// TIA Portal project "Software Units Example - Stack" (V17)

(* hardware
DEVICE "S7-1500/ET200MP station_1"  S7-1500 station
   slot 0: "Rail_0"  Rack  6ES7 590-1***0-0AA0
   slot 1: "PLC_1"  CPU 1515F-2 PN  6ES7 515-2FM01-0AB0  V2.8
      slot 3: "CPU display_1"  6ES7591-1BA00-0AA0
      slot 32768: "PROFINET interface_1"  X1
         slot 32769: "Port_1"  X1 P1
         slot 32770: "Port_2"  X1 P2
      slot 33024: "PROFINET interface_2"  X2
         slot 33025: "Port_1"  X2 P1
      slot 34817: "Virtual CP interface port_1"  Virtual CP interface port  Virtual CP interface port
*)

// ===== PLC "PLC_1"  CPU 1515F-2 PN =====

VAR_GLOBAL   // PLC tag table "Default tag table"
   "System_Byte" AT %MB1 : Byte;
   "FirstScan" AT %M1.0 : Bool;
   "DiagStatusUpdate" AT %M1.1 : Bool;
   "AlwaysTRUE" AT %M1.2 : Bool;
   "AlwaysFALSE" AT %M1.3 : Bool;
   "Clock_Byte" AT %MB0 : Byte;
   "Clock_10Hz" AT %M0.0 : Bool;
   "Clock_5Hz" AT %M0.1 : Bool;
   "Clock_2.5Hz" AT %M0.2 : Bool;
   "Clock_2Hz" AT %M0.3 : Bool;
   "Clock_1.25Hz" AT %M0.4 : Bool;
   "Clock_1Hz" AT %M0.5 : Bool;
   "Clock_0.625Hz" AT %M0.6 : Bool;
   "Clock_0.5Hz" AT %M0.7 : Bool;
END_VAR

VAR_GLOBAL CONSTANT   // PLC tag table "Constants"
   "NULL_TOKEN" : Int := -157;
END_VAR

TYPE "IntStack.UDT"
   STRUCT
      add : DInt;
      data : Array[0..4] of Int;
      length : DInt;
      remove : DInt := 0;
   END_STRUCT;
END_TYPE

TYPE "Stack.Interface.UDT"
   STRUCT
      clear : Bool;
      pop : Bool;
      push : Bool;
      status : String;
      value : Int;
   END_STRUCT;
END_TYPE

DATA_BLOCK "Stack01.Interface.Data"   // DB1
{ S7_Optimized_Access := 'TRUE' }
VERSION : 0.1
BEGIN
END_DATA_BLOCK

DATA_BLOCK "Stack01.Data"   // DB2
{ S7_Optimized_Access := 'TRUE' }
VERSION : 0.1
// stored: InstanceOfName Stack
"Stack"
BEGIN
END_DATA_BLOCK

FUNCTION_BLOCK "Stack"   // FB1, SCL
{ S7_Optimized_Access := 'TRUE' }
VERSION : 0.1
   VAR_IN_OUT
      interface : "Stack.Interface.UDT";
   END_VAR
   VAR
      data : "IntStack.UDT";
   END_VAR
   VAR_TEMP
      blank_interface : "Stack.Interface.UDT";
   END_VAR
BEGIN
   IF #interface.clear THEN
       #interface := #blank_interface;
       #interface.status := "clear"(default_add_index := 0,
                                    default_remove_index := -1,
                                    null_token := "NULL_TOKEN",
                                    buffer := #data);
   END_IF;

   IF #interface.pop THEN
       #interface.pop := FALSE;
       #interface.status := "pop"(null_token := "NULL_TOKEN",
                                  value => #interface.value,
                                  buffer := #data);
   END_IF;

   IF #interface.push THEN
       #interface.push := FALSE;
       #interface.status := "push"(value := #interface.value,
                                   buffer := #data);
       #interface.value := "NULL_TOKEN"; 
   END_IF;
END_FUNCTION_BLOCK

FUNCTION "clear" : String   // FC1, SCL
{ S7_Optimized_Access := 'TRUE' }
AUTHOR : Machado
FAMILY : Int[+]
VERSION : 0.1
   VAR_INPUT
      default_add_index : Int;
      default_remove_index : Int;
      null_token : Int;
   END_VAR
   VAR_IN_OUT
      buffer : "IntStack.UDT";
   END_VAR
   VAR_TEMP
      i : DInt;
      size : DInt;
   END_VAR
   VAR CONSTANT
      DONE : String := 'cleared.';
   END_VAR
BEGIN
   REGION "GET SIZE"
       #size := UDINT_TO_DINT("count_of_elements"(#buffer.data));
   END_REGION

   REGION "CLEAR DATA"
       FOR #i := 0 TO #size - 1 DO
           #buffer.data[#i] := #null_token;
       END_FOR;
   END_REGION

   REGION "CLEAR META DATA"
       #buffer.add := #default_add_index;
       #buffer.remove := #default_remove_index;
       #buffer.length := 0;
   END_REGION

   REGION "RETURN"
       #clear := #DONE;
       RETURN;
   END_REGION
END_FUNCTION

FUNCTION "is_empty" : Bool   // FC2, SCL
TITLE = Int[+] Data Array Is Empty
{ S7_Optimized_Access := 'TRUE' }
AUTHOR : Machado
FAMILY : Int[+]
VERSION : 0.1
// returns true if array is empty
   VAR_INPUT
      buffer : "IntStack.UDT";
   END_VAR
BEGIN
   IF #buffer.length = 0 THEN
       #is_empty := TRUE;
       RETURN;
   END_IF;
   #is_empty := FALSE;
   RETURN;
END_FUNCTION

FUNCTION "pop" : String   // FC3, SCL
{ S7_Optimized_Access := 'TRUE' }
AUTHOR : Machado
FAMILY : Int[+]
VERSION : 0.1
// do not use with Add
   VAR_INPUT
      null_token : Int;
   END_VAR
   VAR_OUTPUT
      value : Int;
   END_VAR
   VAR_IN_OUT
      buffer : "IntStack.UDT";
   END_VAR
   VAR CONSTANT
      ARRAY_EMPTY : String := 'array empty. no operation.';
      POPPED : String := 'popped';
   END_VAR
BEGIN
   REGION "ARRAY EMPTY"
       IF "is_empty"(#buffer) THEN
           #value := #null_token;
           #pop := #ARRAY_EMPTY;
           RETURN;
       END_IF;
   END_REGION


   REGION "POP"
       #value := #buffer.data[#buffer.remove];
       #buffer.data[#buffer.remove] := #null_token;
       #buffer.add -= 1;
       #buffer.remove -= 1;
       #buffer.length -= 1;
       #pop := #POPPED;
       RETURN;
   END_REGION
END_FUNCTION

FUNCTION "is_full" : Bool   // FC4, SCL
TITLE = Array Is Full
{ S7_Optimized_Access := 'TRUE' }
AUTHOR : Machado
FAMILY : Int[+]
VERSION : 0.1
// returns true if array is full
   VAR_INPUT
      buffer : "IntStack.UDT";
   END_VAR
   VAR_TEMP
      size : DInt;
   END_VAR
BEGIN
   #size := UDINT_TO_DINT("count_of_elements"(#buffer.data));
   IF #buffer.length = #size THEN
       #is_full := TRUE;
       RETURN;
   END_IF;
   #is_full := FALSE;
   RETURN;
END_FUNCTION

FUNCTION "push" : String   // FC5, SCL
{ S7_Optimized_Access := 'TRUE' }
AUTHOR : Machado
FAMILY : Int[+]
VERSION : 0.1
// dont use push with remove
   VAR_INPUT
      value : Int;
   END_VAR
   VAR_IN_OUT
      buffer : "IntStack.UDT";
   END_VAR
   VAR CONSTANT
      ARRAY_FULL : String := 'array full. no operation.';
      PUSHED : String := 'pushed.';
   END_VAR
BEGIN
   REGION "ARRAY FULL"
       IF "is_full"(#buffer) THEN
           #push := #ARRAY_FULL;
           RETURN;
       END_IF;
   END_REGION


   REGION "PUSH"
       #buffer.data[#buffer.add] := #value;
       #buffer.add += 1;
       #buffer.remove += 1;
       #buffer.length += 1;
       #push := #PUSHED;
       RETURN;
   END_REGION
END_FUNCTION

FUNCTION "count_of_elements" : UDInt   // FC6, SCL
{ S7_Optimized_Access := 'TRUE' }
VERSION : 0.1
   VAR_INPUT
      data : Variant;
   END_VAR
BEGIN
   #count_of_elements := CountOfElements(#data);
   RETURN;
END_FUNCTION

ORGANIZATION_BLOCK "Main"   // OB1, LAD, ProgramCycle
TITLE = "Main Program Sweep (Cycle)"
{ S7_Optimized_Access := 'TRUE' }
VERSION : 0.1
   VAR_INPUT
      Initial_Call : Bool;   // Initial call of this OB
      Remanence : Bool;   // =True, if remanent data are available
   END_VAR
BEGIN
END_ORGANIZATION_BLOCK

ORGANIZATION_BLOCK "AppOB"   // OB123, SCL, ProgramCycle
TITLE = "Main Program Sweep (Cycle)"
{ S7_Optimized_Access := 'TRUE' }
VERSION : 0.1
   VAR_INPUT
      Initial_Call : Bool;   // Initial call of this OB
      Remanence : Bool;   // =True, if remanent data are available
   END_VAR
BEGIN
   "Stack01.Data"("Stack01.Interface.Data");
END_ORGANIZATION_BLOCK